# EPICS substitutions: hls_pss/testApp/Db/userHost.substitutions
# Example substitutions file

file "db/dbExample1.db" {
    { user = "iocHost" }
}

file db/dbExample2.db {
    pattern { user, no, scan }
        { "iocHost", 1, "1 second" }
        { "iocHost", 2, "2 second" }
        { "iocHost", 3, "5 second" }
}
